FUNCTION_BLOCK FB_Pressure
VAR_INPUT
	IN_1 : BOOL :=TRUE;
	IN_2 : BOOL :=TRUE;
	
END_VAR
VAR_OUTPUT
	Interlock : BOOL;
END_VAR

Interlock := IN_1 AND IN_2;

METHOD Control : BOOL
VAR_IN_OUT
	structure : ST_Pressure;
END_VAR
structure.IN_1St := IN_1;
structure.IN_2St := IN_2;
structure.InterlockSt := Interlock;
END_METHOD

END_FUNCTION_BLOCK

(* stored: Version 1.1.0.1, ProductVersion 3.1.4024.12
   POU FB_Pressure: Id {72f1ff6f-5ad0-4281-8a39-5087777248b0}, SpecialFunc None
   Method Control: Id {682224f5-42da-4faf-bcae-9f57ba126053} *)
